// TIA Portal V19 export
FUNCTION_BLOCK "HOUR"   // FB2, LAD
{ S7_Optimized_Access := 'TRUE' }
// stored: MemoryReserve 100, SetENOAutomatically false
   VAR_INPUT
      "SET TIME" : Int;
      RESET : Bool;
      INPUT : Bool;
   END_VAR
   VAR_OUTPUT
      "PRESENT VALUE OF TIME" : Int;
      DONE : Bool;
   END_VAR
   VAR
      "TIMER 1" { S7_SetPoint := 'True'} : IEC_TIMER;
   END_VAR
   VAR RETAIN
      "COUNTER1 2" { S7_SetPoint := 'True'} : IEC_COUNTER;
      "COUNTER1 1" { S7_SetPoint := 'True'} : IEC_COUNTER;
   END_VAR
   VAR
      BIT { ExternalAccessible := 'False'; ExternalVisible := 'False'; ExternalWritable := 'False'} : Bool;
   END_VAR
   VAR_TEMP   // added for the SCL form of the ladder/FBD networks
      _w1 : Bool;
      _w2 : Bool;
   END_VAR
BEGIN

REGION Network 1
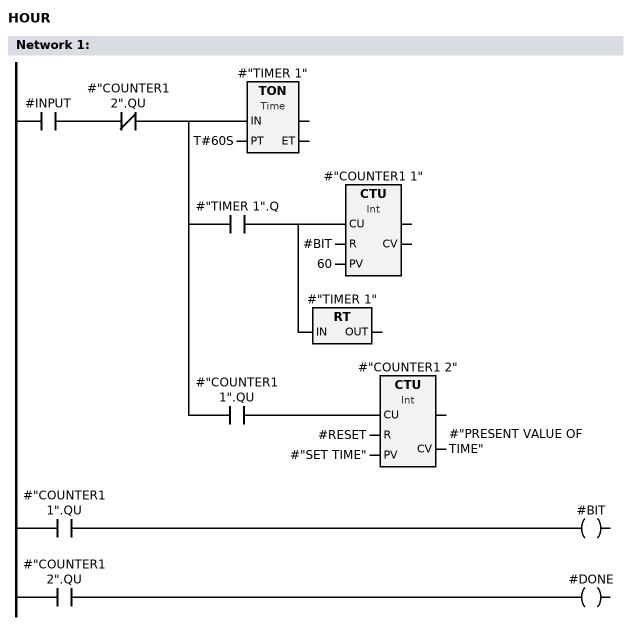
   RUNG wire#powerrail
      Contact( #INPUT )
      I_Contact( #"COUNTER1 2".QU )
      wire#w1
      { S7_Templates := "time_type := Time" } #"TIMER 1".TON(pt := T#60S, et =>)
   END_RUNG
   RUNG wire#w1
      Contact( #"TIMER 1".Q )
      wire#w2
      { S7_Templates := "value_type := Int" } #"COUNTER1 1".CTU(r := #BIT, pv := 60, cv =>)
   END_RUNG
   RUNG wire#w2
      RT_Coil( #"TIMER 1" )
   END_RUNG
   RUNG wire#w1
      Contact( #"COUNTER1 1".QU )
      { S7_Templates := "value_type := Int" } #"COUNTER1 2".CTU(r := #RESET, pv := #"SET TIME", cv => #"PRESENT VALUE OF TIME")
   END_RUNG
   RUNG wire#powerrail
      Contact( #"COUNTER1 1".QU )
      Coil( #BIT )
   END_RUNG
   RUNG wire#powerrail
      Contact( #"COUNTER1 2".QU )
      Coil( #DONE )
   END_RUNG
   // the same network as SCL:
   #_w1 := #INPUT AND NOT #"COUNTER1 2".QU;
   #"TIMER 1".TON(IN := #_w1, PT := T#60S);
   #_w2 := #_w1 AND #"TIMER 1".Q;
   #"COUNTER1 1".CTU(CU := #_w2, R := #BIT, PV := 60);
   IF #_w2 THEN RESET_TIMER(#"TIMER 1"); END_IF;
   #"COUNTER1 2".CTU(CU := #_w1 AND #"COUNTER1 1".QU,
                     R := #RESET,
                     PV := #"SET TIME",
                     CV => #"PRESENT VALUE OF TIME");
   #BIT := #"COUNTER1 1".QU;
   #DONE := #"COUNTER1 2".QU;
END_REGION
END_FUNCTION_BLOCK
